// TIA Portal V19 export
DATA_BLOCK "ALARM DB"   // DB9
{ S7_Optimized_Access := 'TRUE' }
// stored: MemoryReserve 100
   VAR
      "EMG STOP" : Bool;
      "PHASE FAIL" : Bool;
      "AIR PRESSURE FAIL" : Bool;
      "SYRUP MFG VESSEL BOTTOM STERROR TRIP" : Bool;
      "PREMIXING VESSEL BOTTOM STERROR TRIP" : Bool;
      "INLINE 1 HOMOGENIZER MOTOR1 TRIP" : Bool;
      "INLINE 2 HOMOGENIZER MOTOR 2 TRIP" : Bool;
      "FILTER PRESS MOTOR 1 TRIP" : Bool;
      "FILTER PRESS MOTOR 2 TRIP" : Bool;
      "VACCUM PUMP MOTOR 1 TRIP" : Bool;
      "VACCUMP PUMP MOTOR 2 TRIP" : Bool;
      "VACCUMP PUMP MOTOR 3 TRIP" : Bool;
      "VACCUMP PUMP MOTOR 4 TRIP" : Bool;
      "SUGAR VESSEL BOTTOM STERROR TRIP" : Bool;
      "BASKET FILTER MOTOR TRIP" : Bool;
      "SYRUP FLOW SWITCH" : Bool;
      "PREMIXING FLOW SWITCH" : Bool;
      "SUGAR FLOW SWITCH" : Bool;
      "INLINE 1 FLOW SWITCH" : Bool;
      "INLINE 2 FLOW SWITCH" : Bool;
      "MFG TO STORAGE-1 WITH INLINE HOMOGENIZER TRANSFER COMPLETE" : Bool;
      "MFG TO STORAGE-1 WITH FILTER PRESS TRANSFER COMPLETE" : Bool;
      "MFG TO STORAGE-2 WITH INLINE HOMOGENIZER TRANSFER COMPLETE" : Bool;
      "MFG TO STORAGE-2 WITH FILTER PRESS TRANSFER COMPLETE" : Bool;
      "MFG TO STORAGE-3 WITH INLINE HOMOGENIZER TRANSFER COMPLETE" : Bool;
      "MFG TO STORAGE-3 WITH FILTER PRESS TRANSFER COMPLETE" : Bool;
      "PREMIXING TRANSFER COMPLETE" : Bool;
      "SUGAR TRANSFER COMPLETE" : Bool;
   END_VAR
BEGIN
END_DATA_BLOCK
